(* Schneider Machine Expert - Basic project ProjectUPDATRE, file version 2.7.0.0 *)
(* ProjectInformations: Name=New project *)

HARDWARE
  Cpu 0: TM221CE24U
  EthernetConfiguration: NetworkName=M221, IpAllocationMode=ByDhcp, IpAddress=192.168.1.11, SubnetMask=255.255.255.0
  SerialLineConfiguration: Baud=Baud19200, Parity=ParityEven, DataBits=DataBits8, StopBits=StopBits1, PhysicalMedium=PhysicalMediumRs485, TransmissionMode=TransmissionModeModbusRtu, SlaveId=1, Addressing=SlaveAddressing
  MastTask: UsePeriodScanMode=false, PeriodScan=100
  FastTask: Period=255
  CpuBehavior: StartingMode=StartAsPreviousState, AutoSaveRamOnEeprom=true, WatchdogPeriod=250

SYMBOLS  (address, symbol, comment, settings)
  %M0       START_EMITTER  "EMITTER SENT"
  %M1       STOP_EMO
  %M2       SENSOR_START_MAIN
  %M3       SENSOR_STOP_MAIN  "EMITTER"
  %M4       SENSOR_START_CONBLUE1
  %M5       SENSOR_STOP_CONBLUE1
  %M6       SENBLUEINSTOP
  %M7       SENBLUEIN
  %M8       SENCONBLUE2
  %M16      LIM0
  %M17      LIM90
  %M18      BL
  %M19      FL
  %M20      SEN14
  %M21      SECLECTOR_1
  %M22      SECLECTOR_2
  %M23      SEN15
  %M29      SEN16
  %M37        "Grab"
  %M46      DETECT
  %M131     TRUN
  %M132     ROLL_UP
  %M133     ROLL_DN
  %M136     ROLL4
  %M137     ROLL6
  %M139     LIFT
  %M140     CRANE_R
  %M141     CRANE_L
  %M155     BELT_CON62
  %M156     PUSH1
  %M157     PUSH2
  %M162     R2_CLAMP
  %M163     R1_CLAMP
  %M164     R1_RAISE
  %M165     TAP_X
  %M166     TAP_Y
  %M167     TAP_GRAB
  %M311     FULL
  %S0       SB_COLDSTART  "Indicates or executes a cold start (data initialized to default values)"
  %S6       SB_TB1S  "Time base of 1 s generated by an internal clock"
  %MW0      VISION
  %MW1      WEIGHTBLUE
  %MW5      VS2
  %MW6      VS3
  %TM0        [Preset=1, Base=OneSecond]
  %TM1        [Preset=2, Base=OneSecond]
  %TM2        [Type=TOF, Preset=1, Base=OneSecond]
  %TM3        [Preset=1, Base=OneSecond]
  %TM4        [Type=TOF, Preset=12, Base=OneSecond]
  %TM5        [Type=TOF, Preset=15]
  %TM6        [Preset=2, Base=OneSecond]
  %TM7        [Preset=1, Base=OneSecond]
  %TM8        [Preset=2, Base=OneSecond]
  %TM9        [Preset=3, Base=OneSecond]
  %TM10       [Preset=1, Base=OneSecond]
  %TM11       [Preset=2, Base=OneSecond]
  %TM12       [Preset=2, Base=OneSecond]
  %TM13       [Preset=1, Base=OneSecond]
  %TM14       [Preset=1, Base=OneSecond]
  %TM15       [Preset=10, Base=OneHundredMilliSeconds]
  %TM16       [Preset=10, Base=OneHundredMilliSeconds]
  %TM17       [Preset=1, Base=OneSecond]
  %TM18       [Preset=10, Base=OneHundredMilliSeconds]
  %TM19       [Preset=10, Base=OneHundredMilliSeconds]
  %C0         [Preset=0]
  %C1         [Preset=2]
  %C2         [Preset=54]

POU New POU
  (* SectionNumber=1 *)

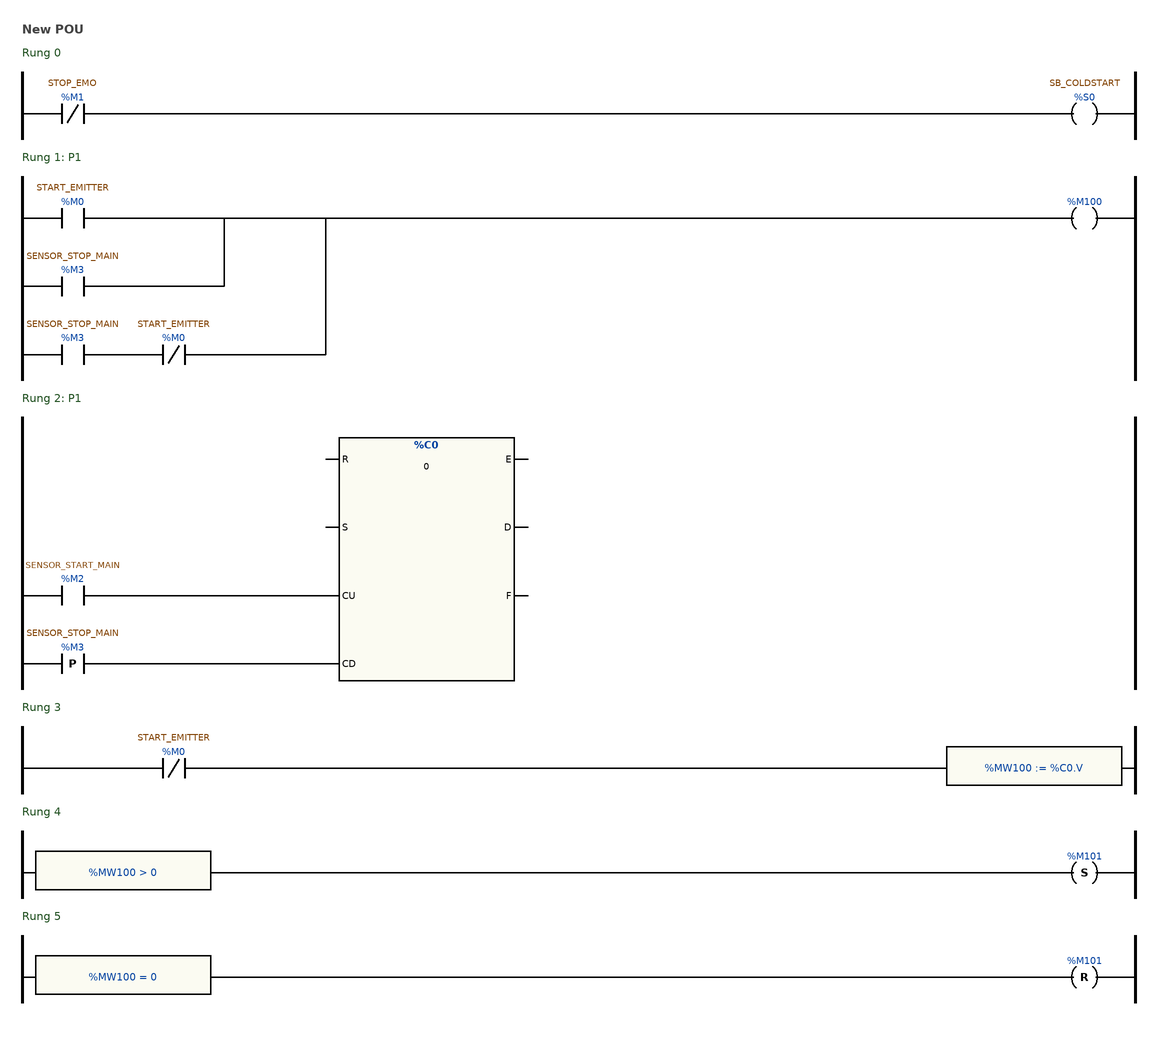

// Rung 0
  LDN %M1                 (* STOP_EMO *)
  ST %S0                  (* SB_COLDSTART *)
  // as ST:
  //   SB_COLDSTART := NOT STOP_EMO;

// Rung 1: P1
  LD %M0                  (* START_EMITTER *)
  OR %M3                  (* SENSOR_STOP_MAIN *)
  OR( %M3                 (* SENSOR_STOP_MAIN *)
  ANDN %M0                (* START_EMITTER *)
  )
  ST %M100
  // as ST:
  //   %M100 := START_EMITTER OR SENSOR_STOP_MAIN OR SENSOR_STOP_MAIN AND NOT START_EMITTER;

// Rung 2: P1
  BLK %C0
  LD %M2                  (* SENSOR_START_MAIN *)
  CU
  LDR %M3                 (* SENSOR_STOP_MAIN *)
  CD
  END_BLK
  // as ST:
  //   %C0(CU := SENSOR_START_MAIN, CD := RISING(SENSOR_STOP_MAIN));

// Rung 3
  LDN %M0                 (* START_EMITTER *)
  [ %MW100 := %C0.V ]
  // as ST:
  //   IF NOT START_EMITTER THEN %MW100 := %C0.V; END_IF;

// Rung 4
  LD [ %MW100 > 0 ]
  S %M101
  // as ST:
  //   IF %MW100 > 0 THEN %M101 := TRUE; END_IF;

// Rung 5
  LD [ %MW100 = 0 ]
  R %M101
  // as ST:
  //   IF %MW100 = 0 THEN %M101 := FALSE; END_IF;

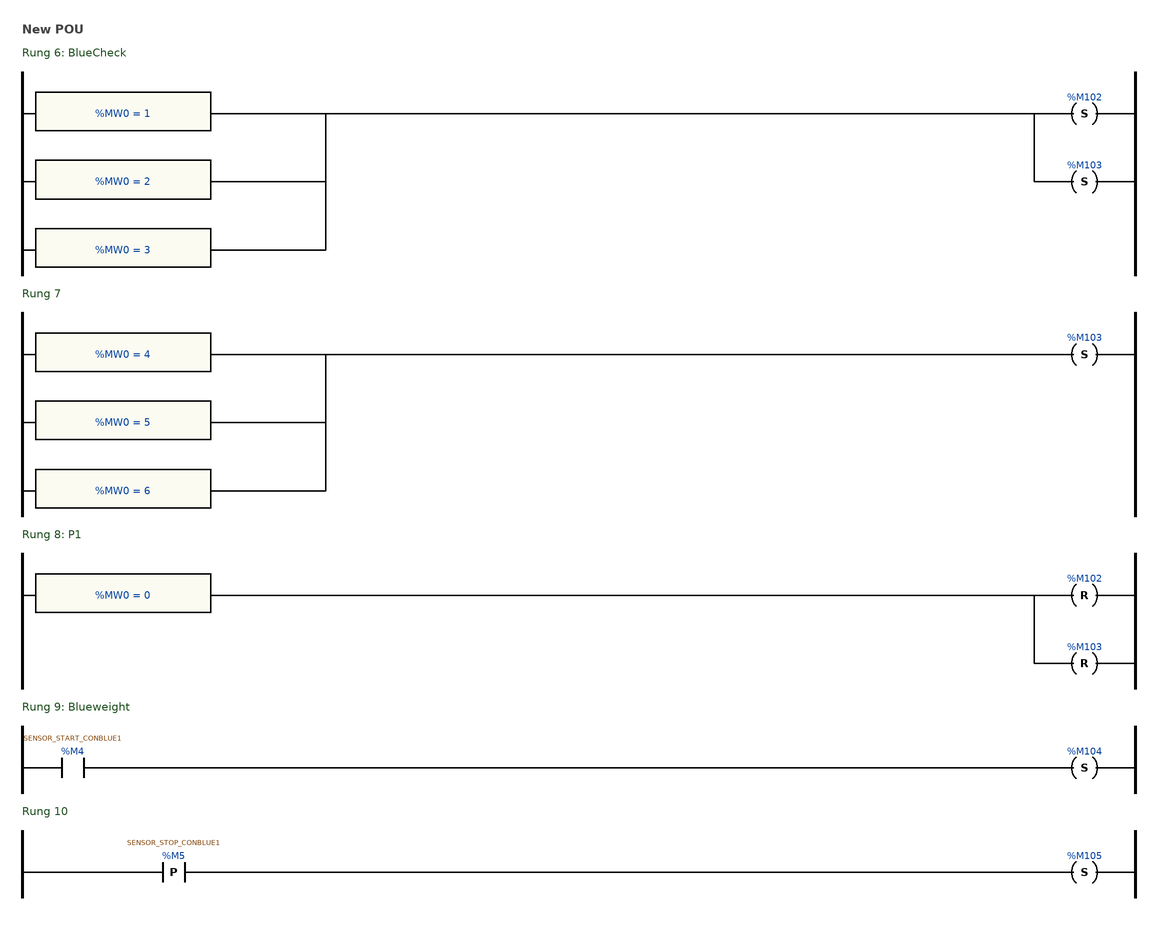

// Rung 6: BlueCheck
  LD [ %MW0 = 1 ]         (* VISION *)
  OR [ %MW0 = 2 ]         (* VISION *)
  OR [ %MW0 = 3 ]         (* VISION *)
  S %M102
  S %M103
  // as ST:
  //   IF VISION = 1 OR VISION = 2 OR VISION = 3 THEN %M102 := TRUE; END_IF;
  //   IF VISION = 1 OR VISION = 2 OR VISION = 3 THEN %M103 := TRUE; END_IF;

// Rung 7
  LD [ %MW0 = 4 ]         (* VISION *)
  OR [ %MW0 = 5 ]         (* VISION *)
  OR [ %MW0 = 6 ]         (* VISION *)
  S %M103
  // as ST:
  //   IF VISION = 4 OR VISION = 5 OR VISION = 6 THEN %M103 := TRUE; END_IF;

// Rung 8: P1
  LD [ %MW0 = 0 ]         (* VISION *)
  R %M102
  R %M103
  // as ST:
  //   IF VISION = 0 THEN %M102 := FALSE; END_IF;
  //   IF VISION = 0 THEN %M103 := FALSE; END_IF;

// Rung 9: Blueweight
  LD %M4                  (* SENSOR_START_CONBLUE1 *)
  S %M104
  // as ST:
  //   IF SENSOR_START_CONBLUE1 THEN %M104 := TRUE; END_IF;

// Rung 10
  LDR %M5                 (* SENSOR_STOP_CONBLUE1 *)
  S %M105
  // as ST:
  //   IF RISING(SENSOR_STOP_CONBLUE1) THEN %M105 := TRUE; END_IF;

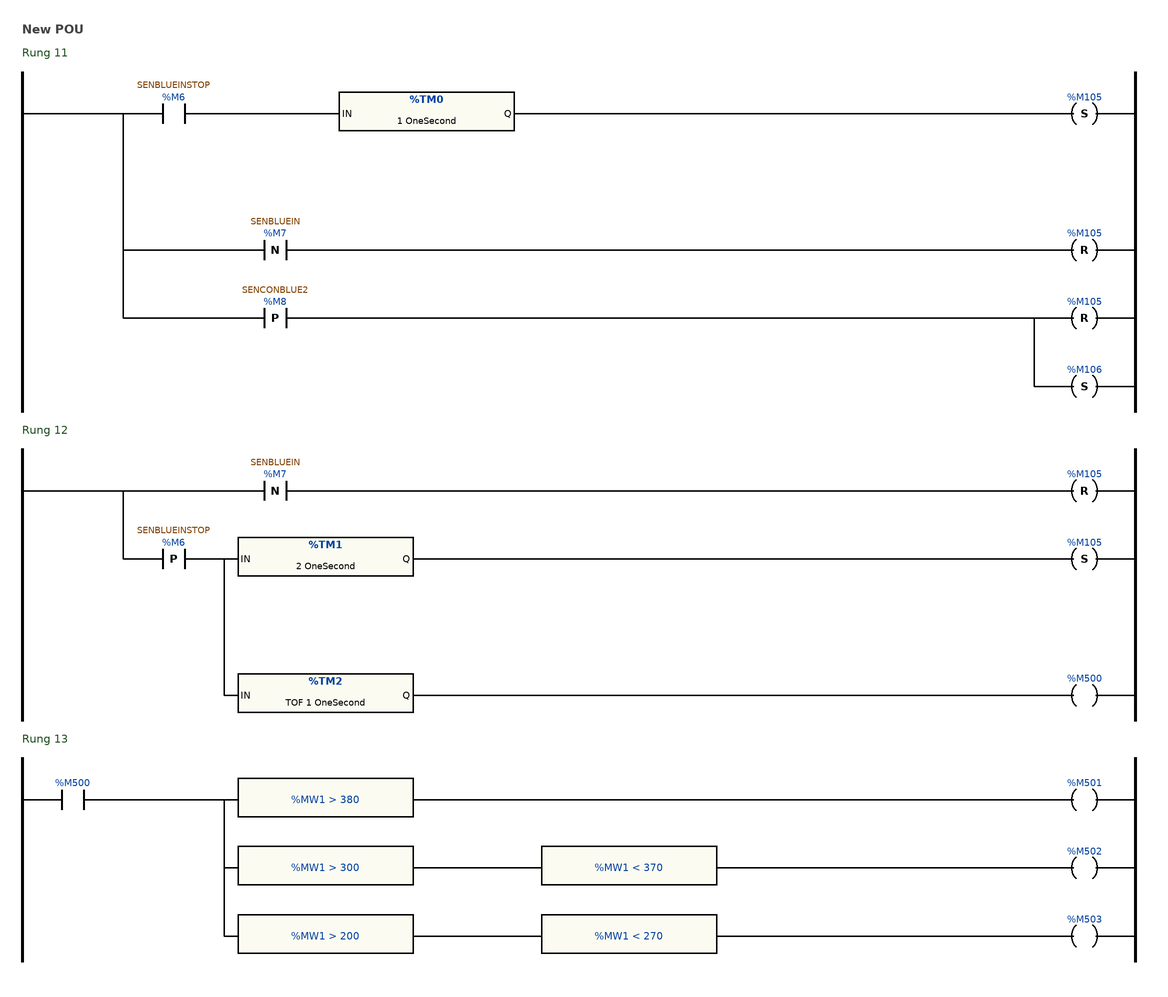

// Rung 11
  LD 1
  MULTIFB
  LD 1
  ST %MW2009:X0
  BLK %TM0
  LD %MW2009:X0
  AND %M6                 (* SENBLUEINSTOP *)
  IN
  OUT_BLK
  LD Q
  S %M105
  END_BLK
  LD %MW2009:X0
  MPS
  ANDF %M7                (* SENBLUEIN *)
  R %M105
  MPP
  ANDR %M8                (* SENCONBLUE2 *)
  R %M105
  S %M106
  MULTIFB
  // as ST:
  //   %TM0(IN := SENBLUEINSTOP);
  //   IF %TM0.Q THEN %M105 := TRUE; END_IF;
  //   IF FALLING(SENBLUEIN) THEN %M105 := FALSE; END_IF;
  //   IF RISING(SENCONBLUE2) THEN %M105 := FALSE; END_IF;
  //   IF RISING(SENCONBLUE2) THEN %M106 := TRUE; END_IF;

// Rung 12
  LD 1
  MULTIFB
  LD 1
  ST %MW2009:X0
  LD %MW2009:X0
  ANDF %M7                (* SENBLUEIN *)
  R %M105
  LD %MW2009:X0
  ANDR %M6                (* SENBLUEINSTOP *)
  ST %MW2009:X1
  BLK %TM1
  LD %MW2009:X1
  IN
  OUT_BLK
  LD Q
  S %M105
  END_BLK
  BLK %TM2
  LD %MW2009:X1
  IN
  OUT_BLK
  LD Q
  ST %M500
  END_BLK
  MULTIFB
  // as ST:
  //   IF FALLING(SENBLUEIN) THEN %M105 := FALSE; END_IF;
  //   %TM1(IN := RISING(SENBLUEINSTOP));
  //   IF %TM1.Q THEN %M105 := TRUE; END_IF;
  //   %TM2(IN := RISING(SENBLUEINSTOP));
  //   %M500 := %TM2.Q;

// Rung 13
  LD %M500
  MPS
  AND [ %MW1 > 380 ]      (* WEIGHTBLUE *)
  ST %M501
  MRD
  AND [ %MW1 > 300 ]      (* WEIGHTBLUE *)
  AND [ %MW1 < 370 ]      (* WEIGHTBLUE *)
  ST %M502
  MPP
  AND [ %MW1 > 200 ]      (* WEIGHTBLUE *)
  AND [ %MW1 < 270 ]      (* WEIGHTBLUE *)
  ST %M503
  // as ST:
  //   %M501 := %M500 AND WEIGHTBLUE > 380;
  //   %M502 := %M500 AND WEIGHTBLUE > 300 AND WEIGHTBLUE < 370;
  //   %M503 := %M500 AND WEIGHTBLUE > 200 AND WEIGHTBLUE < 270;

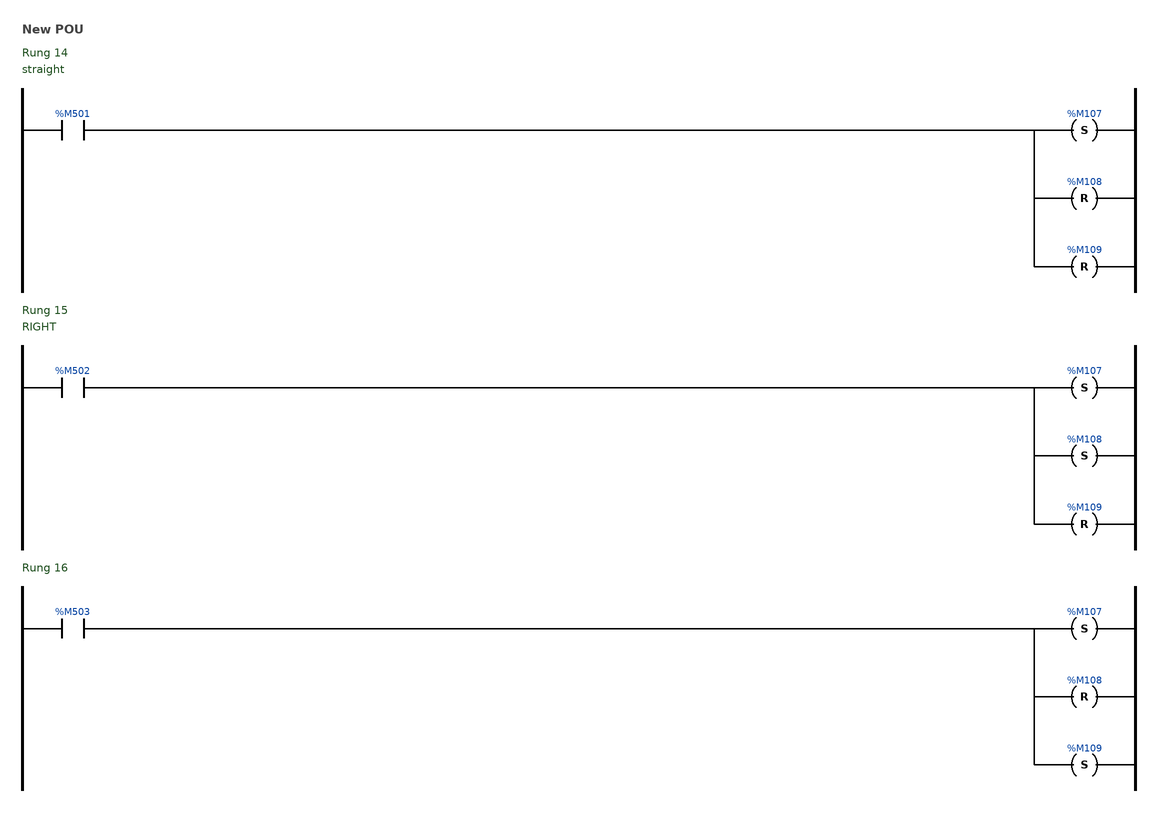

// Rung 14
// straight
  LD %M501
  S %M107
  R %M108
  R %M109
  // as ST:
  //   IF %M501 THEN %M107 := TRUE; END_IF;
  //   IF %M501 THEN %M108 := FALSE; END_IF;
  //   IF %M501 THEN %M109 := FALSE; END_IF;

// Rung 15
// RIGHT
  LD %M502
  S %M107
  S %M108
  R %M109
  // as ST:
  //   IF %M502 THEN %M107 := TRUE; END_IF;
  //   IF %M502 THEN %M108 := TRUE; END_IF;
  //   IF %M502 THEN %M109 := FALSE; END_IF;

// Rung 16
  LD %M503
  S %M107
  R %M108
  S %M109
  // as ST:
  //   IF %M503 THEN %M107 := TRUE; END_IF;
  //   IF %M503 THEN %M108 := FALSE; END_IF;
  //   IF %M503 THEN %M109 := TRUE; END_IF;

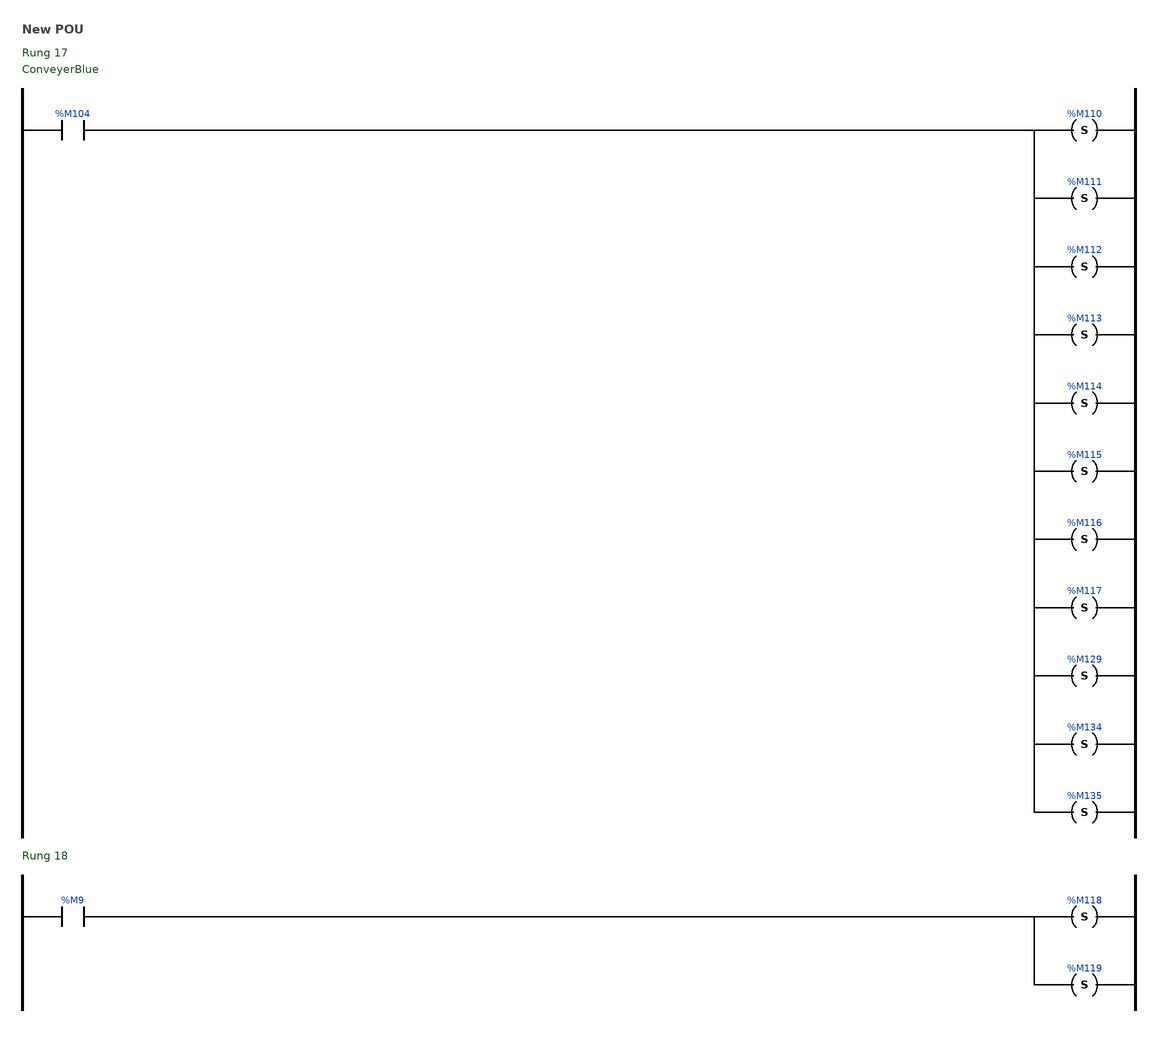

// Rung 17
// ConveyerBlue
  LD %M104
  S %M110
  S %M111
  S %M112
  S %M113
  S %M114
  S %M115
  S %M116
  S %M117
  S %M129
  S %M134
  S %M135
  // as ST:
  //   IF %M104 THEN %M110 := TRUE; END_IF;
  //   IF %M104 THEN %M111 := TRUE; END_IF;
  //   IF %M104 THEN %M112 := TRUE; END_IF;
  //   IF %M104 THEN %M113 := TRUE; END_IF;
  //   IF %M104 THEN %M114 := TRUE; END_IF;
  //   IF %M104 THEN %M115 := TRUE; END_IF;
  //   IF %M104 THEN %M116 := TRUE; END_IF;
  //   IF %M104 THEN %M117 := TRUE; END_IF;
  //   IF %M104 THEN %M129 := TRUE; END_IF;
  //   IF %M104 THEN %M134 := TRUE; END_IF;
  //   IF %M104 THEN %M135 := TRUE; END_IF;

// Rung 18
  LD %M9
  S %M118
  S %M119
  // as ST:
  //   IF %M9 THEN %M118 := TRUE; END_IF;
  //   IF %M9 THEN %M119 := TRUE; END_IF;

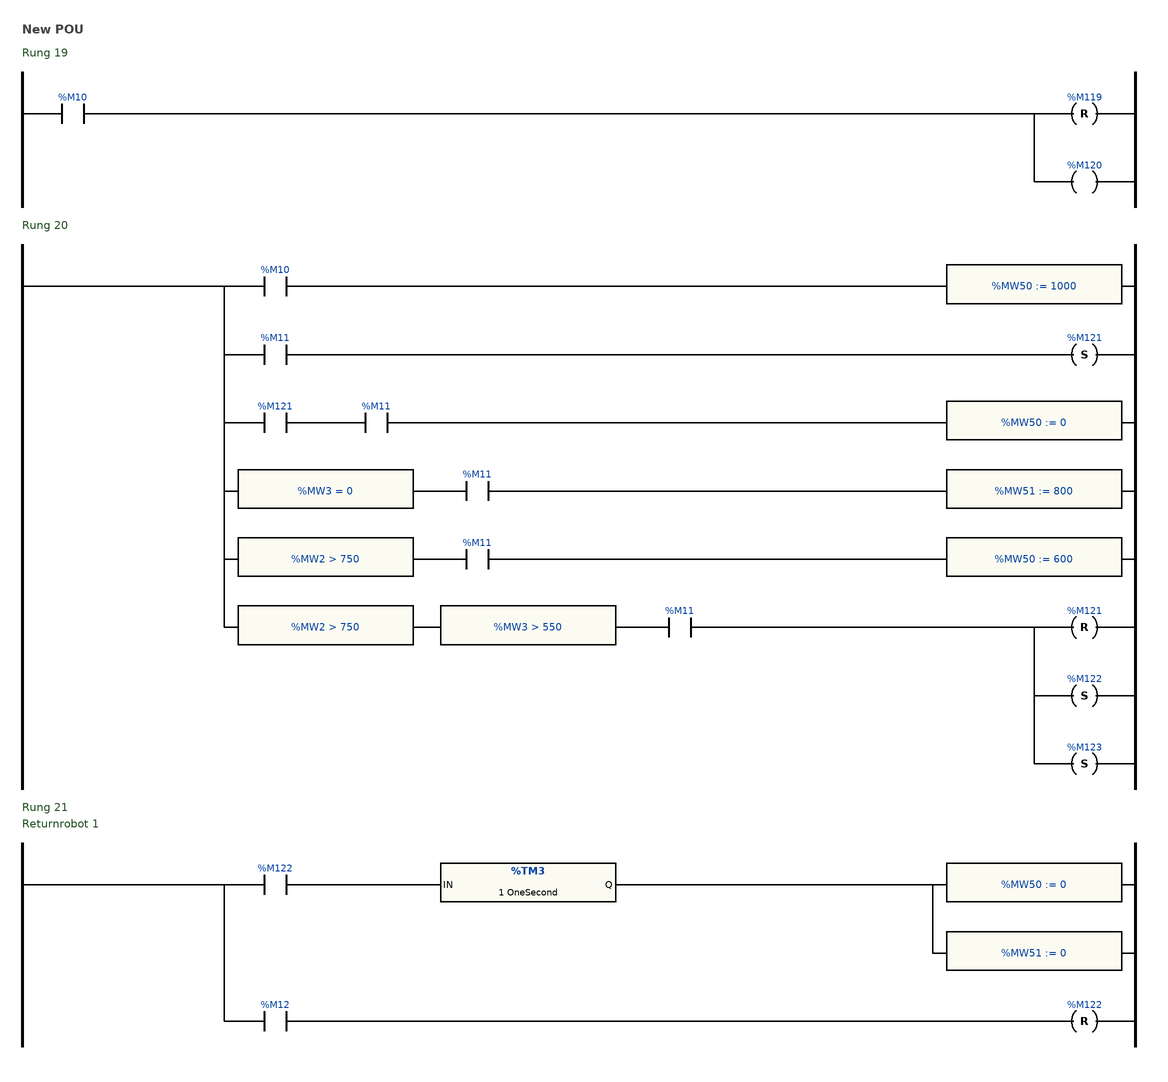

// Rung 19
  LD %M10
  R %M119
  ST %M120
  // as ST:
  //   IF %M10 THEN %M119 := FALSE; END_IF;
  //   %M120 := %M10;

// Rung 20
  LD 1
  MPS
  AND %M10
  [ %MW50 := 1000 ]
  MRD
  AND %M11
  S %M121
  MRD
  AND %M121
  AND %M11
  [ %MW50 := 0 ]
  MRD
  AND [ %MW3 = 0 ]
  AND %M11
  [ %MW51 := 800 ]
  MRD
  AND [ %MW2 > 750 ]
  AND %M11
  [ %MW50 := 600 ]
  MPP
  AND [ %MW2 > 750 ]
  AND [ %MW3 > 550 ]
  AND %M11
  R %M121
  S %M122
  S %M123
  // as ST:
  //   IF %M10 THEN %MW50 := 1000; END_IF;
  //   IF %M11 THEN %M121 := TRUE; END_IF;
  //   IF %M121 AND %M11 THEN %MW50 := 0; END_IF;
  //   IF %MW3 = 0 AND %M11 THEN %MW51 := 800; END_IF;
  //   IF %MW2 > 750 AND %M11 THEN %MW50 := 600; END_IF;
  //   IF %MW2 > 750 AND %MW3 > 550 AND %M11 THEN %M121 := FALSE; END_IF;
  //   IF %MW2 > 750 AND %MW3 > 550 AND %M11 THEN %M122 := TRUE; END_IF;
  //   IF %MW2 > 750 AND %MW3 > 550 AND %M11 THEN %M123 := TRUE; END_IF;

// Rung 21
// Returnrobot 1
  LD 1
  MULTIFB
  LD 1
  ST %MW2009:X0
  BLK %TM3
  LD %MW2009:X0
  AND %M122
  IN
  OUT_BLK
  LD Q
  [ %MW50 := 0 ]
  [ %MW51 := 0 ]
  END_BLK
  LD %MW2009:X0
  AND %M12
  R %M122
  MULTIFB
  // as ST:
  //   %TM3(IN := %M122);
  //   IF %TM3.Q THEN %MW50 := 0; END_IF;
  //   IF %TM3.Q THEN %MW51 := 0; END_IF;
  //   IF %M12 THEN %M122 := FALSE; END_IF;

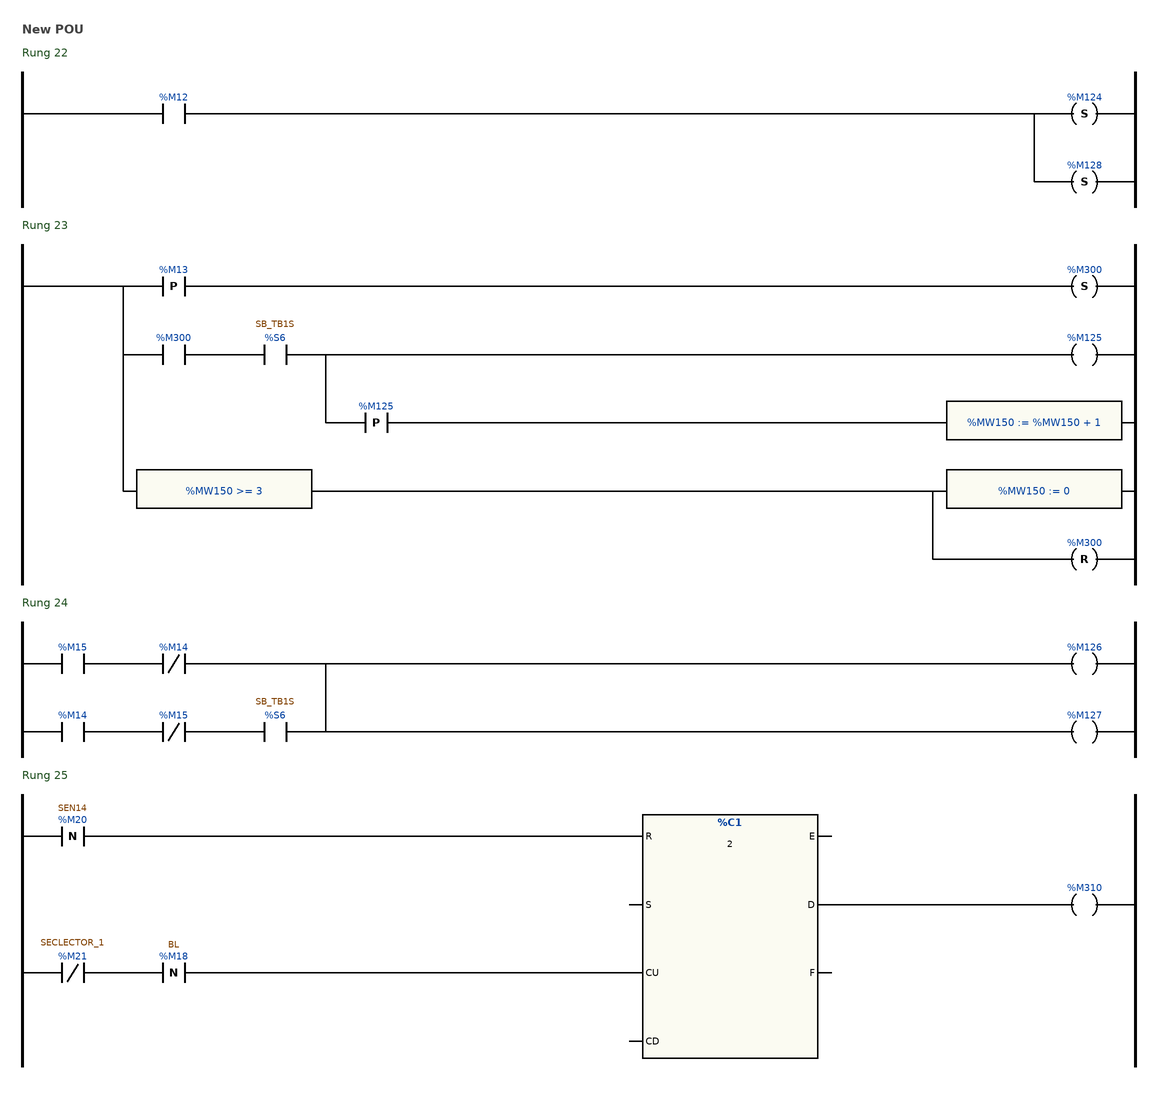

// Rung 22
  LD %M12
  S %M124
  S %M128
  // as ST:
  //   IF %M12 THEN %M124 := TRUE; END_IF;
  //   IF %M12 THEN %M128 := TRUE; END_IF;

// Rung 23
  LD 1
  MPS
  ANDR %M13
  S %M300
  MRD
  AND %M300
  AND %S6                 (* SB_TB1S *)
  MPS
  ST %M125
  MPP
  ANDR %M125
  [ %MW150 := %MW150 + 1 ]
  MPP
  AND [ %MW150 >= 3 ]
  [ %MW150 := 0 ]
  R %M300
  // as ST:
  //   IF RISING(%M13) THEN %M300 := TRUE; END_IF;
  //   %M125 := %M300 AND SB_TB1S;
  //   IF %M300 AND SB_TB1S AND RISING(%M125) THEN %MW150 := %MW150 + 1; END_IF;
  //   _t1 := %MW150 >= 3;
  //   IF _t1 THEN %MW150 := 0; END_IF;
  //   IF _t1 THEN %M300 := FALSE; END_IF;

// Rung 24
  LD %M15
  ANDN %M14
  OR( %M14
  ANDN %M15
  AND %S6                 (* SB_TB1S *)
  )
  ST %M126
  ST %M127
  // as ST:
  //   %M126 := %M15 AND NOT %M14 OR %M14 AND NOT %M15 AND SB_TB1S;
  //   %M127 := %M15 AND NOT %M14 OR %M14 AND NOT %M15 AND SB_TB1S;

// Rung 25
  BLK %C1
  LDF %M20                (* SEN14 *)
  R
  LDN %M21                (* SECLECTOR_1 *)
  ANDF %M18               (* BL *)
  CU
  OUT_BLK
  LD D
  ST %M310
  END_BLK
  // as ST:
  //   %C1(R := FALLING(SEN14), CU := NOT SECLECTOR_1 AND FALLING(BL));
  //   %M310 := %C1.D;

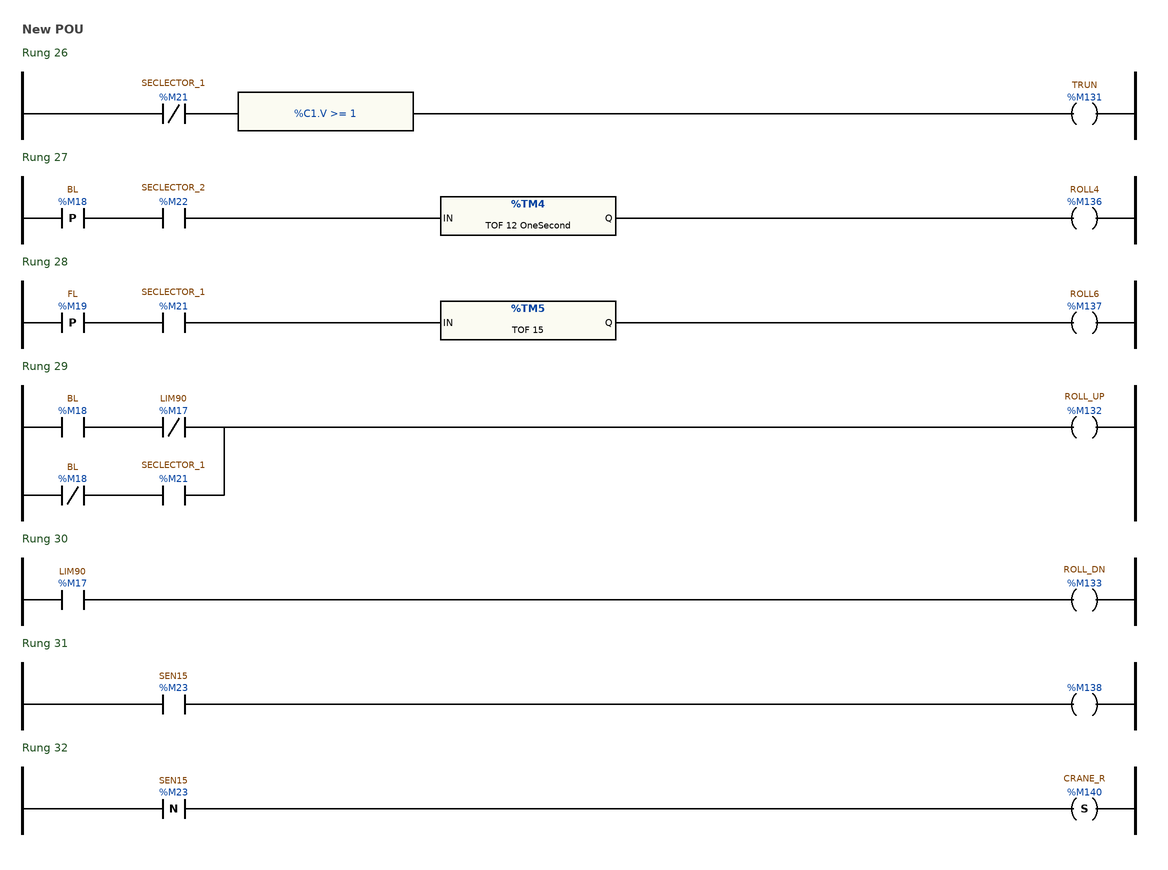

// Rung 26
  LDN %M21                (* SECLECTOR_1 *)
  AND [ %C1.V >= 1 ]
  ST %M131                (* TRUN *)
  // as ST:
  //   TRUN := NOT SECLECTOR_1 AND %C1.V >= 1;

// Rung 27
  BLK %TM4
  LDR %M18                (* BL *)
  AND %M22                (* SECLECTOR_2 *)
  IN
  OUT_BLK
  LD Q
  ST %M136                (* ROLL4 *)
  END_BLK
  // as ST:
  //   %TM4(IN := RISING(BL) AND SECLECTOR_2);
  //   ROLL4 := %TM4.Q;

// Rung 28
  BLK %TM5
  LDR %M19                (* FL *)
  AND %M21                (* SECLECTOR_1 *)
  IN
  OUT_BLK
  LD Q
  ST %M137                (* ROLL6 *)
  END_BLK
  // as ST:
  //   %TM5(IN := RISING(FL) AND SECLECTOR_1);
  //   ROLL6 := %TM5.Q;

// Rung 29
  LD %M18                 (* BL *)
  ANDN %M17               (* LIM90 *)
  OR(N %M18               (* BL *)
  AND %M21                (* SECLECTOR_1 *)
  )
  ST %M132                (* ROLL_UP *)
  // as ST:
  //   ROLL_UP := BL AND NOT LIM90 OR NOT BL AND SECLECTOR_1;

// Rung 30
  LD %M17                 (* LIM90 *)
  ST %M133                (* ROLL_DN *)
  // as ST:
  //   ROLL_DN := LIM90;

// Rung 31
  LD %M23                 (* SEN15 *)
  ST %M138
  // as ST:
  //   %M138 := SEN15;

// Rung 32
  LDF %M23                (* SEN15 *)
  S %M140                 (* CRANE_R *)
  // as ST:
  //   IF FALLING(SEN15) THEN CRANE_R := TRUE; END_IF;

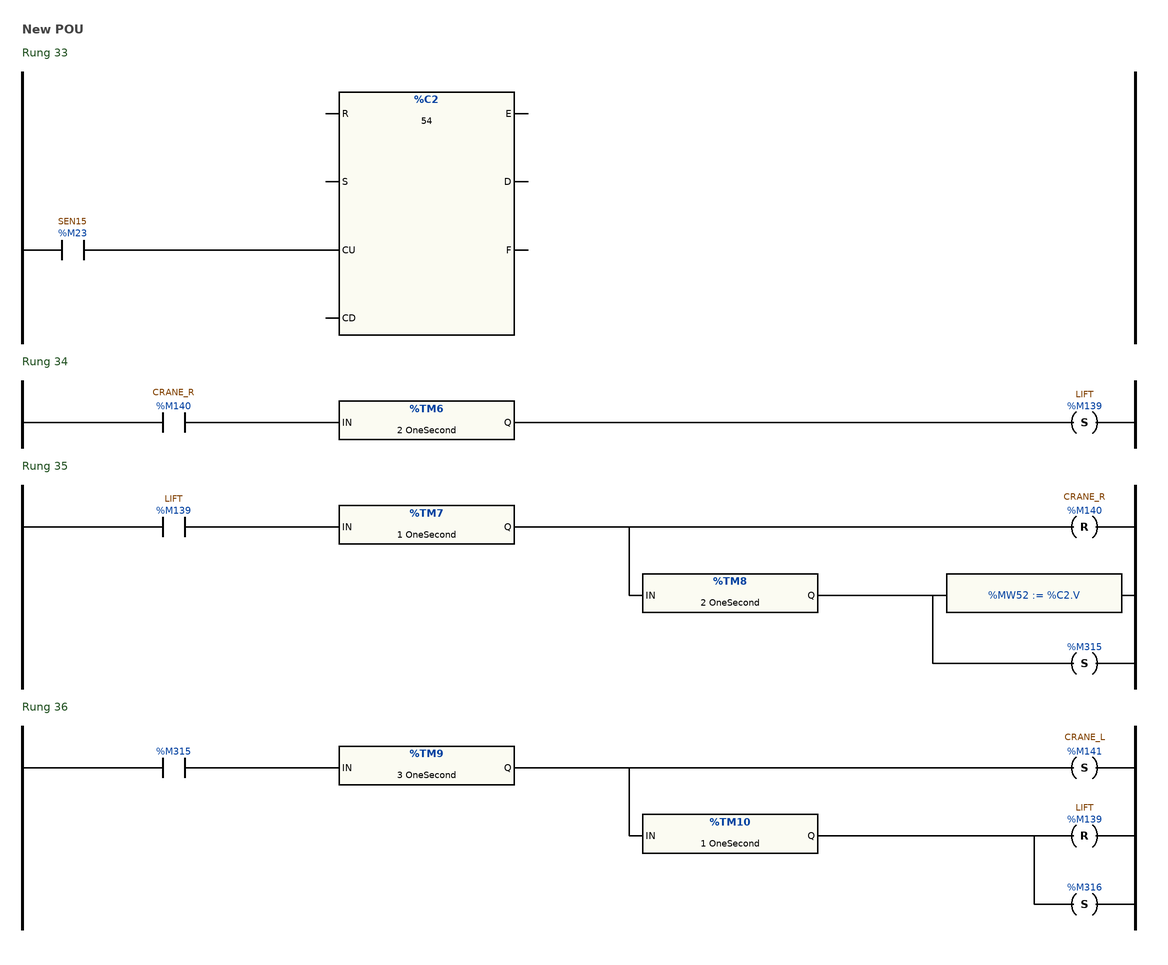

// Rung 33
  BLK %C2
  LD %M23                 (* SEN15 *)
  CU
  END_BLK
  // as ST:
  //   %C2(CU := SEN15);

// Rung 34
  BLK %TM6
  LD %M140                (* CRANE_R *)
  IN
  OUT_BLK
  LD Q
  S %M139                 (* LIFT *)
  END_BLK
  // as ST:
  //   %TM6(IN := CRANE_R);
  //   IF %TM6.Q THEN LIFT := TRUE; END_IF;

// Rung 35
  LD 1
  MULTIFB
  BLK %TM7
  LD 1
  AND %M139               (* LIFT *)
  IN
  OUT_BLK
  LD Q
  ST %MW2009:X0
  END_BLK
  LD %MW2009:X0
  R %M140                 (* CRANE_R *)
  BLK %TM8
  LD %MW2009:X0
  IN
  OUT_BLK
  LD Q
  [ %MW52 := %C2.V ]
  S %M315
  END_BLK
  MULTIFB
  // as ST:
  //   %TM7(IN := LIFT);
  //   IF %TM7.Q THEN CRANE_R := FALSE; END_IF;
  //   %TM8(IN := %TM7.Q);
  //   IF %TM8.Q THEN %MW52 := %C2.V; END_IF;
  //   IF %TM8.Q THEN %M315 := TRUE; END_IF;

// Rung 36
  LD 1
  MULTIFB
  BLK %TM9
  LD 1
  AND %M315
  IN
  OUT_BLK
  LD Q
  ST %MW2009:X0
  END_BLK
  LD %MW2009:X0
  S %M141                 (* CRANE_L *)
  BLK %TM10
  LD %MW2009:X0
  IN
  OUT_BLK
  LD Q
  R %M139                 (* LIFT *)
  S %M316
  END_BLK
  MULTIFB
  // as ST:
  //   %TM9(IN := %M315);
  //   IF %TM9.Q THEN CRANE_L := TRUE; END_IF;
  //   %TM10(IN := %TM9.Q);
  //   IF %TM10.Q THEN LIFT := FALSE; END_IF;
  //   IF %TM10.Q THEN %M316 := TRUE; END_IF;

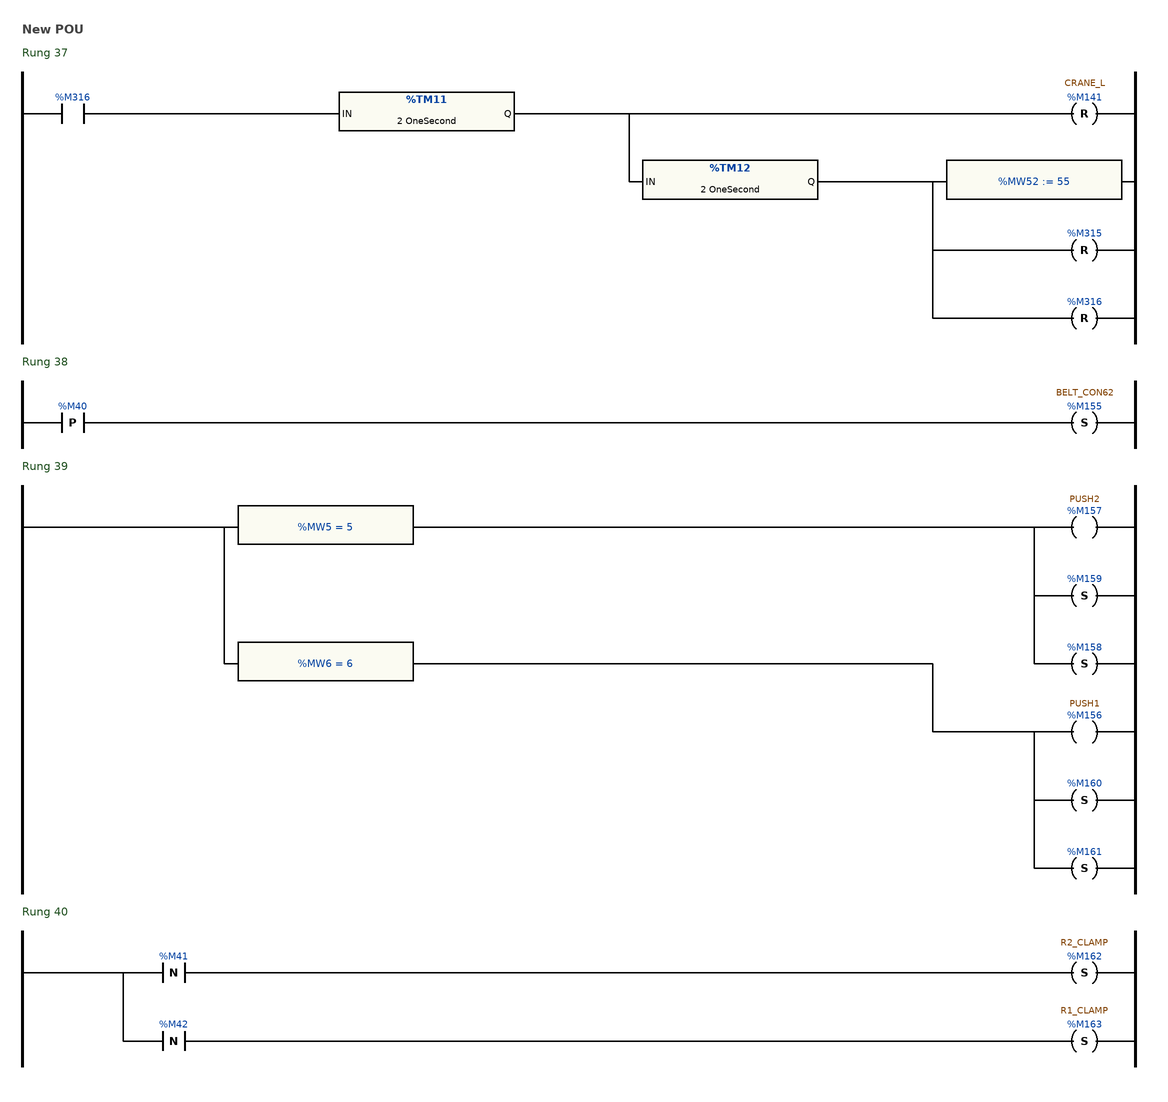

// Rung 37
  LD 1
  MULTIFB
  BLK %TM11
  LD 1
  AND %M316
  IN
  OUT_BLK
  LD Q
  ST %MW2009:X0
  END_BLK
  LD %MW2009:X0
  R %M141                 (* CRANE_L *)
  BLK %TM12
  LD %MW2009:X0
  IN
  OUT_BLK
  LD Q
  [ %MW52 := 55 ]
  R %M315
  R %M316
  END_BLK
  MULTIFB
  // as ST:
  //   %TM11(IN := %M316);
  //   IF %TM11.Q THEN CRANE_L := FALSE; END_IF;
  //   %TM12(IN := %TM11.Q);
  //   IF %TM12.Q THEN %MW52 := 55; END_IF;
  //   IF %TM12.Q THEN %M315 := FALSE; END_IF;
  //   IF %TM12.Q THEN %M316 := FALSE; END_IF;

// Rung 38
  LDR %M40
  S %M155                 (* BELT_CON62 *)
  // as ST:
  //   IF RISING(%M40) THEN BELT_CON62 := TRUE; END_IF;

// Rung 39
  LD 1
  MPS
  AND [ %MW5 = 5 ]        (* VS2 *)
  ST %M157                (* PUSH2 *)
  S %M159
  S %M158
  MPP
  AND [ %MW6 = 6 ]        (* VS3 *)
  ST %M156                (* PUSH1 *)
  S %M160
  S %M161
  // as ST:
  //   PUSH2 := VS2 = 5;
  //   IF VS2 = 5 THEN %M159 := TRUE; END_IF;
  //   IF VS2 = 5 THEN %M158 := TRUE; END_IF;
  //   PUSH1 := VS3 = 6;
  //   IF VS3 = 6 THEN %M160 := TRUE; END_IF;
  //   IF VS3 = 6 THEN %M161 := TRUE; END_IF;

// Rung 40
  LD 1
  MPS
  ANDF %M41
  S %M162                 (* R2_CLAMP *)
  MPP
  ANDF %M42
  S %M163                 (* R1_CLAMP *)
  // as ST:
  //   IF FALLING(%M41) THEN R2_CLAMP := TRUE; END_IF;
  //   IF FALLING(%M42) THEN R1_CLAMP := TRUE; END_IF;

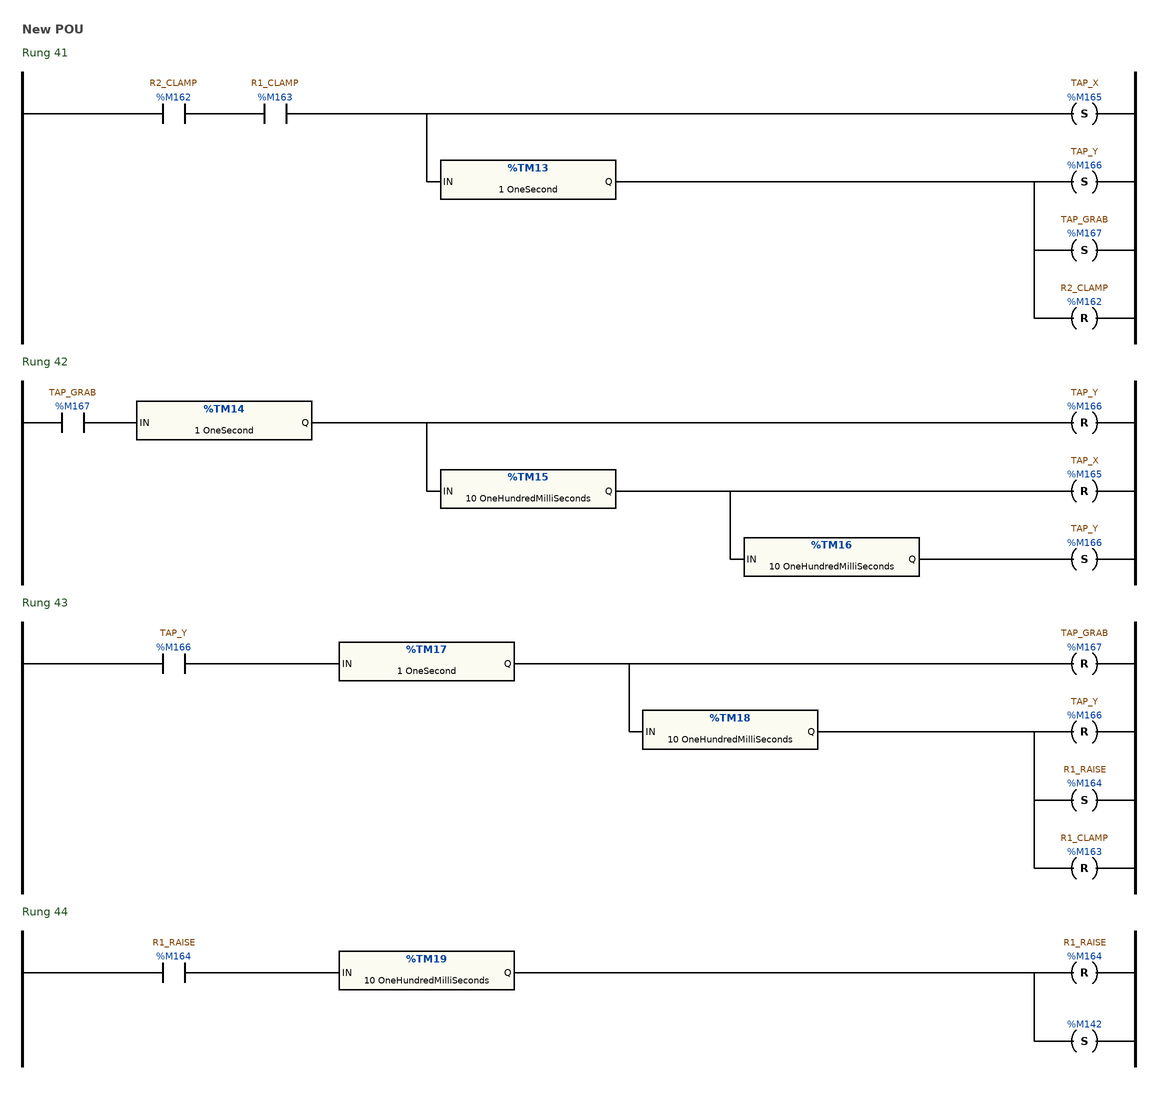

// Rung 41
  LD 1
  MULTIFB
  LD 1
  AND %M162               (* R2_CLAMP *)
  AND %M163               (* R1_CLAMP *)
  ST %MW2009:X0
  LD %MW2009:X0
  S %M165                 (* TAP_X *)
  BLK %TM13
  LD %MW2009:X0
  IN
  OUT_BLK
  LD Q
  S %M166                 (* TAP_Y *)
  S %M167                 (* TAP_GRAB *)
  R %M162                 (* R2_CLAMP *)
  END_BLK
  MULTIFB
  // as ST:
  //   IF R2_CLAMP AND R1_CLAMP THEN TAP_X := TRUE; END_IF;
  //   %TM13(IN := R2_CLAMP AND R1_CLAMP);
  //   IF %TM13.Q THEN TAP_Y := TRUE; END_IF;
  //   IF %TM13.Q THEN TAP_GRAB := TRUE; END_IF;
  //   IF %TM13.Q THEN R2_CLAMP := FALSE; END_IF;

// Rung 42
  LD 1
  MULTIFB
  BLK %TM14
  LD 1
  AND %M167               (* TAP_GRAB *)
  IN
  OUT_BLK
  LD Q
  ST %MW2009:X0
  END_BLK
  LD %MW2009:X0
  R %M166                 (* TAP_Y *)
  BLK %TM15
  LD %MW2009:X0
  IN
  OUT_BLK
  LD Q
  ST %MW2009:X1
  END_BLK
  LD %MW2009:X1
  R %M165                 (* TAP_X *)
  BLK %TM16
  LD %MW2009:X1
  IN
  OUT_BLK
  LD Q
  S %M166                 (* TAP_Y *)
  END_BLK
  MULTIFB
  // as ST:
  //   %TM14(IN := TAP_GRAB);
  //   IF %TM14.Q THEN TAP_Y := FALSE; END_IF;
  //   %TM15(IN := %TM14.Q);
  //   IF %TM15.Q THEN TAP_X := FALSE; END_IF;
  //   %TM16(IN := %TM15.Q);
  //   IF %TM16.Q THEN TAP_Y := TRUE; END_IF;

// Rung 43
  LD 1
  MULTIFB
  BLK %TM17
  LD 1
  AND %M166               (* TAP_Y *)
  IN
  OUT_BLK
  LD Q
  ST %MW2009:X0
  END_BLK
  LD %MW2009:X0
  R %M167                 (* TAP_GRAB *)
  BLK %TM18
  LD %MW2009:X0
  IN
  OUT_BLK
  LD Q
  R %M166                 (* TAP_Y *)
  S %M164                 (* R1_RAISE *)
  R %M163                 (* R1_CLAMP *)
  END_BLK
  MULTIFB
  // as ST:
  //   %TM17(IN := TAP_Y);
  //   IF %TM17.Q THEN TAP_GRAB := FALSE; END_IF;
  //   %TM18(IN := %TM17.Q);
  //   IF %TM18.Q THEN TAP_Y := FALSE; END_IF;
  //   IF %TM18.Q THEN R1_RAISE := TRUE; END_IF;
  //   IF %TM18.Q THEN R1_CLAMP := FALSE; END_IF;

// Rung 44
  BLK %TM19
  LD %M164                (* R1_RAISE *)
  IN
  OUT_BLK
  LD Q
  R %M164                 (* R1_RAISE *)
  S %M142
  END_BLK
  // as ST:
  //   %TM19(IN := R1_RAISE);
  //   IF %TM19.Q THEN R1_RAISE := FALSE; END_IF;
  //   IF %TM19.Q THEN %M142 := TRUE; END_IF;

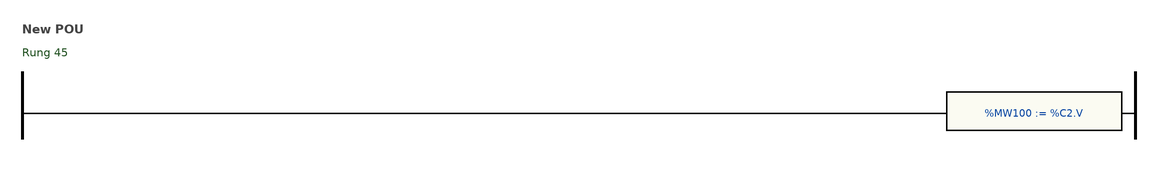

// Rung 45
  LD 1
  [ %MW100 := %C2.V ]
  // as ST:
  //   %MW100 := %C2.V;
